FUNCTION_BLOCK MOD_InputBelt
VAR_INPUT
	i_InputSensor 	: MOD_InputBelt_I_stSensor;
	i_OutputSensor 	: MOD_InputBelt_I_stSensor;
END_VAR
VAR_OUTPUT
	q_NewBox 		: MOD_InputBelt_Q_stRequest;
	q_BeltMotorOn 	: MOD_InputBelt_Q_stMotor := (MoveLeft := FALSE, MoveRight := FALSE);
	q_BoxReady 		: MOD_InputBelt_Q_stOutput;
END_VAR
VAR_IN_OUT
	iq_CommandState : INT;
END_VAR
VAR
	State 			: INT := 10;
	Executing 		: BOOL := FALSE;//variable for main state. used for orderly code
END_VAR

CASE iq_CommandState OF
	Command.Abort:
		q_BeltMotorOn.MoveLeft 	:= FALSE;
		Executing 				:= FALSE;
		
	Command.Executing:
		Executing 				:= TRUE;
		
	Command.Hold:
		Executing 				:= FALSE;
		q_BeltMotorOn.MoveLeft 	:= FALSE;
		
	Command.Reset:
		Executing 				:= FALSE;
		State 					:= 10;//reset state
		q_BeltMotorOn.MoveLeft 	:= FALSE;
		
	Command.Stop:		
		IF State = 20 THEN
			Executing 				:= FALSE;
			q_BeltMotorOn.MoveLeft 	:= FALSE;
		ELSE
			Executing 				:= TRUE;			
		END_IF		
END_CASE

IF Executing THEN
CASE State OF
	10://startup //reset?
		IF i_InputSensor.Blocked = TRUE AND i_OutputSensor.Blocked = TRUE THEN
			State := 11;
		ELSIF i_InputSensor.Blocked = FALSE AND i_OutputSensor.Blocked = FALSE THEN
			State := 20;
		ELSIF i_InputSensor.Blocked = TRUE AND i_OutputSensor.Blocked = FALSE THEN
			State := 30;
		ELSIF i_InputSensor.Blocked = FALSE AND i_OutputSensor.Blocked = TRUE THEN
			State := 40;		
		END_IF
		
	11://startup boxes on belt.
		q_NewBox.NewBox 		:= FALSE;
		q_BeltMotorOn.MoveLeft 	:= FALSE;
		q_BoxReady.BoxReady 	:= TRUE;
	
		IF i_OutputSensor.Blocked = FALSE THEN
			State := 20;
		END_IF
		
	20://No Box
		q_NewBox.NewBox 		:= TRUE;
		q_BeltMotorOn.MoveLeft 	:= FALSE;
		q_BoxReady.BoxReady 	:= FALSE;
		
		IF i_InputSensor.Blocked = TRUE AND i_OutputSensor.Blocked = FALSE THEN
			State := 30;
		END_IF
	
	30://retrieve box
		q_NewBox.NewBox 		:= FALSE;
		q_BeltMotorOn.MoveLeft 	:= TRUE;
		q_BoxReady.BoxReady 	:= FALSE;
		
		IF i_InputSensor.Blocked = FALSE AND i_OutputSensor.Blocked = TRUE THEN
			State := 40;
		END_IF
		
	40://boxready
		q_NewBox.NewBox 		:= FALSE;
		q_BeltMotorOn.MoveLeft 	:= FALSE;
		q_BoxReady.BoxReady 	:= TRUE;
		
		IF i_OutputSensor.Blocked = FALSE THEN
			State := 20;
		END_IF

END_CASE
END_IF

END_FUNCTION_BLOCK

(* stored: Version 1.1.0.1, ProductVersion 3.1.4024.6
   POU MOD_InputBelt: Id {2a85e218-1bdb-4ed5-9bd6-698ec9057a87}, SpecialFunc None *)
